{region '#Template'}
	{attribute 'Version' := '5.0.0.0'}
	{attribute 'Tags' := '"LCID": "1031", "Text": "Universal, Sensor, BI, BV"'}
	{attribute 'Tags' := '"LCID": "1033", "Text": "Universal, Sensor, BI, BV"'}
	{attribute 'Using' := '"Type": "Template", "URI": "EC_ID"'}
	{attribute 'Using' := '"Type": "Template", "URI": "BA2_Param"'}
	{attribute 'Description' := '"LCID": "1031", "Text": "Kombination aus BV BI"'}
	{attribute 'Description' := '"LCID": "1033", "Text": "Combination of BV BI"'}
{endregion}	 
FUNCTION_BLOCK FB_BA_CombinationBI_BV EXTENDS FB_BA_View
VAR_INPUT
END_VAR
VAR_INPUT CONSTANT
	Input				: FB_BA_BI_Raw;	
	Value				: FB_BA_BV_Op;									
END_VAR
VAR_OUTPUT
	bBI_PrVal			: BOOL;
	bTrigBI_PrVal		: BOOL;	
	bBV_PrVal			: BOOL;
	bTrigBV_PrVal		: BOOL;		
END_VAR
VAR
	TrigInput			: FB_BA_RFTrig;
	TrigValue			: FB_BA_RFTrig;
END_VAR

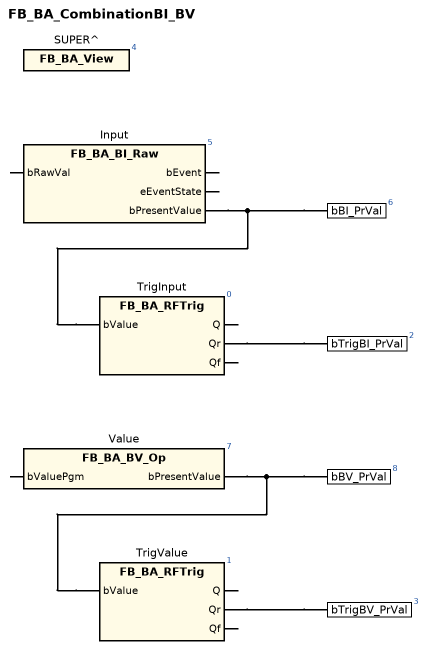
TrigInput(bValue := Input.bPresentValue); // FB_BA_RFTrig
TrigValue(bValue := Value.bPresentValue); // FB_BA_RFTrig
bTrigBI_PrVal := TrigInput.Qr;
bTrigBV_PrVal := TrigValue.Qr;
SUPER^(); // FB_BA_View
Input(); // FB_BA_BI_Raw
bBI_PrVal := Input.bPresentValue;
Value(); // FB_BA_BV_Op
bBV_PrVal := Value.bPresentValue;

METHOD FB_init : BOOL
VAR_INPUT
	bInitRetains : BOOL; // if TRUE, the retain variables are initialized (warm start / cold start)
	bInCopyCode : BOOL;  // if TRUE, the instance afterwards gets moved into the copy code (online change)
END_VAR
Input.iParent						:= THIS^;
Input.iLabel						:= LblFun_Button; 
Input.ePolarity						:= E_BA_Polarity.eReverse;
Input.sActiveText 					:= txtEvent_On;
Input.sInactiveText 				:= txtEvent_Off;
Input.nEventClassID					:= EC_ID.NC80;
Input.stTimeDelay.nToNormal			:= BA2_Param.nDefTimeDelay_ToNormal;
Input.stTimeDelay.nToAbnormal		:= BA2_Param.nDefTimeDelay_ToAbnormal;
Input.bAlarmValue					:= TRUE;
Input.aEventTransitionText[1]		:= txtEvent_Off;
Input.aEventTransitionText[2]		:= txtEvent_None;
Input.aEventTransitionText[3]		:= txtEvent_On;
Input.bEventDetectionEnable			:= FALSE;
Input.eEnPlantLock					:= E_BA_LockPriority.eNoLock;	

Value.iParent						:= THIS^;		
Value.iLabel						:= LblFun_Button; 
Value.sActiveText					:= txtEvent_On;
Value.sInactiveText					:= txtEvent_Off;
Value.bValueRm						:= FALSE;
Value.eToggleMode 					:= E_BA_ToggleMode.eSwitch;
END_METHOD

END_FUNCTION_BLOCK

(* stored: Version 1.1.0.1, ProductVersion 3.1.4024.12
   POU FB_BA_CombinationBI_BV: Id {98e9f744-4293-4233-80b6-efdc769e5bcd}, SpecialFunc None
   Method FB_init: Id {62af4ccf-a83f-474b-92f1-193c092f017d} *)
